(* PLC project Generated.project, CODESYS CODESYS V3.5 SP19 Patch 1 *)
(* stored: creationDateTime 2026-08-11T18:19:14.808468, modificationDateTime 2026-08-11T18:19:14.808468 *)

(* ═══════════════════════════════════════════════════════════════ 🎚️ ST_Modes_Autorisations — Bus d'autorisations du mode machine ─────────────────────────────────────────────────────────────── 📄 Doc métier : DOC/AF/AF_Partie-05_Modes_Maintenance_v2.0.md DOC/AF/AF_Partie-02_Architecture_Programme_v3.1.md §2 🎯 Produit par FB_Modes (via PRG_MODES_CFC) Consommé par : Cycle, Safety, Treuils, Translation, Supervision, Acquisition 🎯 Producteur unique : FB_Modes (via PRG_MODES_CFC) ═══════════════════════════════════════════════════════════════ *)
TYPE ST_Modes_Autorisations : STRUCT
  Mode : E_Mode;  (* Mode arbitré (DISABLE/N1/N2/SEMI_AUTO) *)
  SyncEnable : BOOL;  (* Synchro M1/M2 (logique positive) *)
  InhibitM1 : BOOL;  (* Inhibition M1 (MAINT_N2 only) *)
  InhibitM2 : BOOL;  (* Inhibition M2 (MAINT_N2 only) *)
  JoystickWinchSelectArbitrated : INT;  (* 0=M1+M2 couplés nominal, 1=M1, 2=M2 (unitaires MAINT_N2) *)
  HomingApproachEnable : BOOL;  (* Dépassement butée haut (N2) *)
  MaintenanceM3TargetEnable : BOOL;  (* Cible Translation Maintenance (N2 only) *)
END_STRUCT;
END_TYPE

(* values of E_Mode: DISABLE: Mode Désactivé / Veille de sécurité (sorties bloquées); MAINT_N1: Manuel Niveau 1 : Pilotage unitaire avec toutes sécurités actives; MAINT_N2: Manuel Niveau 2 : Pilotage dégradé (droits étendus + bypasses autorisés); SEMI_AUTO: Mode Semi-Automatique (séquenceur automatique) *)

{attribute 'qualified_only'}
{attribute 'strict'}
TYPE E_Mode : (DISABLE := 0, MAINT_N1 := 1, MAINT_N2 := 2, SEMI_AUTO := 3);
END_TYPE
